// TIA Portal V16 export
// export: Created 2022-01-12T14:32:04.6959631Z, ExportSetting WithDefaults, DisplayName Totally Integrated Automation Portal, DisplayVersion V16 Update 4, DisplayName TIA Portal Version Control Interface, DisplayVersion V16 Update 2, DisplayName TIA Portal Openness, DisplayVersion V16 Update 4, DisplayName STEP 7 Professional, DisplayVersion V16 Update 4, DisplayName STEP 7 Safety, DisplayVersion V16, DisplayName WinCC Professional, DisplayVersion V16 Update 4
DATA_BLOCK "Cip"   // DB8
VERSION : 0.1
// stored: AutoNumber true, DBAccessibleFromOPCUA true, InstanceOfName FB_obsluga_obiektow, InstanceOfType FB
"FB_obsluga_obiektow"
   // VAR
   //    obiekt : Array[0..110] of "typObiekt";
   //    tor : Array[0..2] of "typFunkcjeObiektówCipu";
   //    x { ExternalAccessible := 'False'; ExternalVisible := 'False'; ExternalWritable := 'False'} : Int := 111;
   // END_VAR
BEGIN
   obiekt[0].typObiektu := 0;
   obiekt[1..11].typObiektu := 5;
   obiekt[12..13].typObiektu := 12;
   obiekt[14..20].typObiektu := 18;
   obiekt[21..22].typObiektu := 2;
   obiekt[23..30].typObiektu := 1;
   obiekt[31..32].typObiektu := 4;
   obiekt[33..41].typObiektu := 1;
   obiekt[42..44].typObiektu := 9;
   obiekt[45..49].typObiektu := 1;
   obiekt[50..53].typObiektu := 9;
   obiekt[54..58].typObiektu := 1;
   obiekt[59..62].typObiektu := 9;
   obiekt[63..68].typObiektu := 1;
   obiekt[69..71].typObiektu := 9;
   obiekt[72..78].typObiektu := 1;
   obiekt[79..82].typObiektu := 9;
   obiekt[83..87].typObiektu := 1;
   obiekt[88..90].typObiektu := 9;
   obiekt[91..93].typObiektu := 1;
   obiekt[94..96].typObiektu := 9;
   obiekt[97..98].typObiektu := 4;
   obiekt[99..100].typObiektu := 3;
   obiekt[101..105].typObiektu := 9;
   obiekt[106..107].typObiektu := 17;
   obiekt[108..110].typObiektu := 1;
   obiekt[0].nazwaObiektu := 'C2W1LL01';
   obiekt[1].nazwaObiektu := 'C2W1TT01';
   obiekt[2].nazwaObiektu := 'C2R1TT01';
   obiekt[3].nazwaObiektu := 'C2L1TT01';
   obiekt[4].nazwaObiektu := 'C2A1TT01';
   obiekt[5].nazwaObiektu := 'C2D1TT01';
   obiekt[6].nazwaObiektu := 'C2D2TT01';
   obiekt[7].nazwaObiektu := 'C2D3TT01';
   obiekt[8].nazwaObiektu := 'C211TT01';
   obiekt[9].nazwaObiektu := 'C212TT01';
   obiekt[10].nazwaObiektu := 'C201TT01';
   obiekt[11].nazwaObiektu := 'C202TT01';
   obiekt[12].nazwaObiektu := 'C212QIC01';
   obiekt[13].nazwaObiektu := 'C211QIC01';
   obiekt[14].nazwaObiektu := 'C2A1LT01';
   obiekt[15].nazwaObiektu := 'C2D1LT01';
   obiekt[16].nazwaObiektu := 'C2D2LT01';
   obiekt[17].nazwaObiektu := 'C2D3LT01';
   obiekt[18].nazwaObiektu := 'C2L1LT01';
   obiekt[19].nazwaObiektu := 'C2R1LT01';
   obiekt[20].nazwaObiektu := 'C2W1LT01';
   obiekt[21..22].nazwaObiektu := 'C202CV21';
   obiekt[23].nazwaObiektu := 'C201AV01';
   obiekt[24].nazwaObiektu := 'C201AV02';
   obiekt[25].nazwaObiektu := 'C201AV21';
   obiekt[26].nazwaObiektu := 'C202AV01';
   obiekt[27].nazwaObiektu := 'C202AV02';
   obiekt[28].nazwaObiektu := 'C202AV03';
   obiekt[29].nazwaObiektu := 'C202AV04';
   obiekt[30].nazwaObiektu := 'C202AV21';
   obiekt[31].nazwaObiektu := 'C202FC01';
   obiekt[32].nazwaObiektu := 'C201CP01';
   obiekt[33].nazwaObiektu := 'C211AV01';
   obiekt[34].nazwaObiektu := 'C212AV01';
   obiekt[35].nazwaObiektu := 'C2A1AV01';
   obiekt[36].nazwaObiektu := 'C2A1AV02';
   obiekt[37].nazwaObiektu := 'C2A1AV11';
   obiekt[38].nazwaObiektu := 'C2A1AV12';
   obiekt[39].nazwaObiektu := 'C2A1AV31';
   obiekt[40].nazwaObiektu := 'C2A1AV41';
   obiekt[41].nazwaObiektu := 'C2A1AV42';
   obiekt[42].nazwaObiektu := 'C2A1LH01';
   obiekt[43].nazwaObiektu := 'C2A1LL41';
   obiekt[44].nazwaObiektu := 'C2A1PD01';
   obiekt[45].nazwaObiektu := 'C2D1AV01';
   obiekt[46].nazwaObiektu := 'C2D1AV11';
   obiekt[47].nazwaObiektu := 'C2D1AV41';
   obiekt[48].nazwaObiektu := 'C2D1AV42';
   obiekt[49].nazwaObiektu := 'C2D1AV81';
   obiekt[50].nazwaObiektu := 'C2D1LH01';
   obiekt[51].nazwaObiektu := 'C2D1LL01';
   obiekt[52].nazwaObiektu := 'C2D1LL81';
   obiekt[53].nazwaObiektu := 'C2D1PD01';
   obiekt[54].nazwaObiektu := 'C2D2AV01';
   obiekt[55].nazwaObiektu := 'C2D2AV11';
   obiekt[56].nazwaObiektu := 'C2D2AV41';
   obiekt[57].nazwaObiektu := 'C2D2AV42';
   obiekt[58].nazwaObiektu := 'C2D2AV81';
   obiekt[59].nazwaObiektu := 'C2D2LH01';
   obiekt[60].nazwaObiektu := 'C2D2LL01';
   obiekt[61].nazwaObiektu := 'C2D2LL81';
   obiekt[62].nazwaObiektu := 'C2D2PD01';
   obiekt[63].nazwaObiektu := 'C2D3AV01';
   obiekt[64].nazwaObiektu := 'C2D3AV11';
   obiekt[65].nazwaObiektu := 'C2D3AV31';
   obiekt[66].nazwaObiektu := 'C2D3AV41';
   obiekt[67].nazwaObiektu := 'C2D3AV42';
   obiekt[68].nazwaObiektu := 'C2D3AV43';
   obiekt[69].nazwaObiektu := 'C2D3LH01';
   obiekt[70].nazwaObiektu := 'C2D3LL01';
   obiekt[71].nazwaObiektu := 'C2D3PD01';
   obiekt[72].nazwaObiektu := 'C2L1AV01';
   obiekt[73].nazwaObiektu := 'C2L1AV02';
   obiekt[74].nazwaObiektu := 'C2L1AV11';
   obiekt[75].nazwaObiektu := 'C2L1AV12';
   obiekt[76].nazwaObiektu := 'C2L1AV31';
   obiekt[77].nazwaObiektu := 'C2L1AV41';
   obiekt[78].nazwaObiektu := 'C2L1AV42';
   obiekt[79].nazwaObiektu := 'C2L1LH01';
   obiekt[80].nazwaObiektu := 'C2L1Ll01';
   obiekt[81].nazwaObiektu := 'C2L1Ll41';
   obiekt[82].nazwaObiektu := 'C2L1PD01';
   obiekt[83].nazwaObiektu := 'C2R1AV01';
   obiekt[84].nazwaObiektu := 'C2R1AV02';
   obiekt[85].nazwaObiektu := 'C2R1AV11';
   obiekt[86].nazwaObiektu := 'C2R1AV12';
   obiekt[87].nazwaObiektu := 'C2R1AV41';
   obiekt[88].nazwaObiektu := 'C2R1LH01';
   obiekt[89].nazwaObiektu := 'C2R1LL01';
   obiekt[90].nazwaObiektu := 'C2R1PD01';
   obiekt[91].nazwaObiektu := 'C2W1AV02';
   obiekt[92].nazwaObiektu := 'C2W1AV31';
   obiekt[93].nazwaObiektu := 'C2W1AV41';
   obiekt[94].nazwaObiektu := 'C2W1LH01';
   obiekt[95].nazwaObiektu := 'C2W1LL01';
   obiekt[96].nazwaObiektu := 'C2W1PD01';
   obiekt[97..98].nazwaObiektu := 'C2D1MP81';
   obiekt[99].nazwaObiektu := 'C2A1MP41';
   obiekt[100].nazwaObiektu := 'C2L1MP41';
   obiekt[101].nazwaObiektu := 'C211FV01';
   obiekt[102].nazwaObiektu := 'C212FV01';
   obiekt[103].nazwaObiektu := 'C2D1FV81';
   obiekt[104].nazwaObiektu := 'C2D2FV81';
   obiekt[105].nazwaObiektu := 'C2A1LL01';
   obiekt[106..107].nazwaObiektu := 'F100AV01';
   obiekt[108].nazwaObiektu := 'C2A1AV43';
   obiekt[109].nazwaObiektu := 'C2L1AV43';
   obiekt[110].nazwaObiektu := 'C2W1AV01';
   obiekt[0..20].procedura := 0;
   obiekt[21].procedura := 3;
   obiekt[22].procedura := 0;
   obiekt[23].procedura := 2;
   obiekt[24].procedura := 1;
   obiekt[25].procedura := 2;
   obiekt[26..28].procedura := 0;
   obiekt[29].procedura := 2;
   obiekt[30].procedura := 0;
   obiekt[31].procedura := 3;
   obiekt[32].procedura := 6;
   obiekt[33].procedura := 2;
   obiekt[34].procedura := 0;
   obiekt[35].procedura := 2;
   obiekt[36].procedura := 0;
   obiekt[37].procedura := 2;
   obiekt[38].procedura := 0;
   obiekt[39].procedura := 2;
   obiekt[40..71].procedura := 0;
   obiekt[72].procedura := 2;
   obiekt[73].procedura := 0;
   obiekt[74].procedura := 2;
   obiekt[75].procedura := 0;
   obiekt[76].procedura := 2;
   obiekt[77..91].procedura := 0;
   obiekt[92].procedura := 2;
   obiekt[93..98].procedura := 0;
   obiekt[99].procedura := 2;
   obiekt[100..109].procedura := 0;
   obiekt[110].procedura := 4;
   obiekt[0..20].inStartAuto := FALSE;
   obiekt[21].inStartAuto := TRUE;
   obiekt[22..23].inStartAuto := FALSE;
   obiekt[24..25].inStartAuto := TRUE;
   obiekt[26..30].inStartAuto := FALSE;
   obiekt[31..32].inStartAuto := TRUE;
   obiekt[33..34].inStartAuto := FALSE;
   obiekt[35].inStartAuto := TRUE;
   obiekt[36..91].inStartAuto := FALSE;
   obiekt[92].inStartAuto := TRUE;
   obiekt[93..110].inStartAuto := FALSE;
   obiekt[0..20].outStartUrządzenie := FALSE;
   obiekt[21].outStartUrządzenie := TRUE;
   obiekt[22..23].outStartUrządzenie := FALSE;
   obiekt[24..25].outStartUrządzenie := TRUE;
   obiekt[26..30].outStartUrządzenie := FALSE;
   obiekt[31..32].outStartUrządzenie := TRUE;
   obiekt[33..34].outStartUrządzenie := FALSE;
   obiekt[35].outStartUrządzenie := TRUE;
   obiekt[36..91].outStartUrządzenie := FALSE;
   obiekt[92].outStartUrządzenie := TRUE;
   obiekt[93..110].outStartUrządzenie := FALSE;
   obiekt[0..110].inLiftUp := FALSE;
   obiekt[0..110].outLiftUp := FALSE;
   obiekt[0..110].inLiftDown := FALSE;
   obiekt[0..110].outLiftDown := FALSE;
   obiekt[0..20].inZadaneWysterowanieAuto := 0.0;
   obiekt[21].inZadaneWysterowanieAuto := 100.0;
   obiekt[22..23].inZadaneWysterowanieAuto := 0.0;
   obiekt[24].inZadaneWysterowanieAuto := 100.0;
   obiekt[25..28].inZadaneWysterowanieAuto := 0.0;
   obiekt[29].inZadaneWysterowanieAuto := 100.0;
   obiekt[30].inZadaneWysterowanieAuto := 0.0;
   obiekt[31..32].inZadaneWysterowanieAuto := 100.0;
   obiekt[33..98].inZadaneWysterowanieAuto := 0.0;
   obiekt[99].inZadaneWysterowanieAuto := 100.0;
   obiekt[100..110].inZadaneWysterowanieAuto := 0.0;
   obiekt[0..20].outWysterowanieUrządzenia := 0.0;
   obiekt[21].outWysterowanieUrządzenia := 100.0;
   obiekt[22..23].outWysterowanieUrządzenia := 0.0;
   obiekt[24].outWysterowanieUrządzenia := 100.0;
   obiekt[25..30].outWysterowanieUrządzenia := 0.0;
   obiekt[31..32].outWysterowanieUrządzenia := 100.0;
   obiekt[33..110].outWysterowanieUrządzenia := 0.0;
   obiekt[0].inJestPotwWysterowania := TRUE;
   obiekt[1..22].inJestPotwWysterowania := FALSE;
   obiekt[23..24].inJestPotwWysterowania := TRUE;
   obiekt[25].inJestPotwWysterowania := FALSE;
   obiekt[26..29].inJestPotwWysterowania := TRUE;
   obiekt[30].inJestPotwWysterowania := FALSE;
   obiekt[31..40].inJestPotwWysterowania := TRUE;
   obiekt[41].inJestPotwWysterowania := FALSE;
   obiekt[42..48].inJestPotwWysterowania := TRUE;
   obiekt[49].inJestPotwWysterowania := FALSE;
   obiekt[50..57].inJestPotwWysterowania := TRUE;
   obiekt[58].inJestPotwWysterowania := FALSE;
   obiekt[59..77].inJestPotwWysterowania := TRUE;
   obiekt[78].inJestPotwWysterowania := FALSE;
   obiekt[79..98].inJestPotwWysterowania := TRUE;
   obiekt[99..100].inJestPotwWysterowania := FALSE;
   obiekt[101..105].inJestPotwWysterowania := TRUE;
   obiekt[106..109].inJestPotwWysterowania := FALSE;
   obiekt[110].inJestPotwWysterowania := TRUE;
   obiekt[0..20].diPotwWysterowania := FALSE;
   obiekt[21].diPotwWysterowania := TRUE;
   obiekt[22..41].diPotwWysterowania := FALSE;
   obiekt[42].diPotwWysterowania := TRUE;
   obiekt[43..49].diPotwWysterowania := FALSE;
   obiekt[50].diPotwWysterowania := TRUE;
   obiekt[51..58].diPotwWysterowania := FALSE;
   obiekt[59].diPotwWysterowania := TRUE;
   obiekt[60..68].diPotwWysterowania := FALSE;
   obiekt[69].diPotwWysterowania := TRUE;
   obiekt[70..77].diPotwWysterowania := FALSE;
   obiekt[78..79].diPotwWysterowania := TRUE;
   obiekt[80..87].diPotwWysterowania := FALSE;
   obiekt[88].diPotwWysterowania := TRUE;
   obiekt[89..93].diPotwWysterowania := FALSE;
   obiekt[94].diPotwWysterowania := TRUE;
   obiekt[95..110].diPotwWysterowania := FALSE;
   obiekt[0..110].inJestPotwNiewysterowania := FALSE;
   obiekt[0..21].diPotwNieWysterowania := FALSE;
   obiekt[22].diPotwNieWysterowania := TRUE;
   obiekt[23..110].diPotwNieWysterowania := FALSE;
   obiekt[0..20].inZezwolenieNaPracę := FALSE;
   obiekt[21..41].inZezwolenieNaPracę := TRUE;
   obiekt[42..44].inZezwolenieNaPracę := FALSE;
   obiekt[45..49].inZezwolenieNaPracę := TRUE;
   obiekt[50..53].inZezwolenieNaPracę := FALSE;
   obiekt[54..58].inZezwolenieNaPracę := TRUE;
   obiekt[59..62].inZezwolenieNaPracę := FALSE;
   obiekt[63..68].inZezwolenieNaPracę := TRUE;
   obiekt[69..71].inZezwolenieNaPracę := FALSE;
   obiekt[72..78].inZezwolenieNaPracę := TRUE;
   obiekt[79..82].inZezwolenieNaPracę := FALSE;
   obiekt[83..87].inZezwolenieNaPracę := TRUE;
   obiekt[88..90].inZezwolenieNaPracę := FALSE;
   obiekt[91..93].inZezwolenieNaPracę := TRUE;
   obiekt[94..96].inZezwolenieNaPracę := FALSE;
   obiekt[97..100].inZezwolenieNaPracę := TRUE;
   obiekt[101..107].inZezwolenieNaPracę := FALSE;
   obiekt[108..110].inZezwolenieNaPracę := TRUE;
   obiekt[0..110].Awaria := FALSE;
   obiekt[0..110].ResetAwaria := FALSE;
   obiekt[0..110].kodBłedu := 16#0000;
   obiekt[0..110].czasDoAwariiSP := 1000;
   obiekt[0..30].czasDoAwariiPV := 0;
   obiekt[31].czasDoAwariiPV := 17;
   obiekt[32..41].czasDoAwariiPV := 0;
   obiekt[42].czasDoAwariiPV := 5;
   obiekt[43..49].czasDoAwariiPV := 0;
   obiekt[50].czasDoAwariiPV := 5;
   obiekt[51..58].czasDoAwariiPV := 0;
   obiekt[59].czasDoAwariiPV := 5;
   obiekt[60..68].czasDoAwariiPV := 0;
   obiekt[69].czasDoAwariiPV := 5;
   obiekt[70..78].czasDoAwariiPV := 0;
   obiekt[79].czasDoAwariiPV := 5;
   obiekt[80..87].czasDoAwariiPV := 0;
   obiekt[88].czasDoAwariiPV := 5;
   obiekt[89..93].czasDoAwariiPV := 0;
   obiekt[94].czasDoAwariiPV := 5;
   obiekt[95..110].czasDoAwariiPV := 0;
   obiekt[0..110].czasPracyGodziny := 0.0;
   obiekt[0..110]._ := FALSE;
   obiekt[0..110].hmiPokażStacyjkę := FALSE;
   obiekt[0].hmiStanUrządzenia := 2;
   obiekt[1..20].hmiStanUrządzenia := 1;
   obiekt[21].hmiStanUrządzenia := 3;
   obiekt[22..23].hmiStanUrządzenia := 1;
   obiekt[24..25].hmiStanUrządzenia := 3;
   obiekt[26..30].hmiStanUrządzenia := 1;
   obiekt[31..32].hmiStanUrządzenia := 3;
   obiekt[33..34].hmiStanUrządzenia := 1;
   obiekt[35].hmiStanUrządzenia := 3;
   obiekt[36..41].hmiStanUrządzenia := 1;
   obiekt[42].hmiStanUrządzenia := 3;
   obiekt[43..49].hmiStanUrządzenia := 1;
   obiekt[50].hmiStanUrządzenia := 3;
   obiekt[51..58].hmiStanUrządzenia := 1;
   obiekt[59].hmiStanUrządzenia := 3;
   obiekt[60..68].hmiStanUrządzenia := 1;
   obiekt[69].hmiStanUrządzenia := 3;
   obiekt[70..78].hmiStanUrządzenia := 1;
   obiekt[79].hmiStanUrządzenia := 3;
   obiekt[80].hmiStanUrządzenia := 4;
   obiekt[81..87].hmiStanUrządzenia := 1;
   obiekt[88].hmiStanUrządzenia := 2;
   obiekt[89].hmiStanUrządzenia := 4;
   obiekt[90..91].hmiStanUrządzenia := 1;
   obiekt[92].hmiStanUrządzenia := 3;
   obiekt[93].hmiStanUrządzenia := 1;
   obiekt[94..95].hmiStanUrządzenia := 2;
   obiekt[96..104].hmiStanUrządzenia := 1;
   obiekt[105].hmiStanUrządzenia := 4;
   obiekt[106..110].hmiStanUrządzenia := 1;
   obiekt[0..110].hmiTrybAutoManual := FALSE;
   obiekt[0..110].hmiManualStart := FALSE;
   obiekt[0..110].hmiManualStop := FALSE;
   obiekt[0..110].hmiManualLiftUp := FALSE;
   obiekt[0..110].hmiManualLiftDown := FALSE;
   obiekt[0..110].hmiManualneWysterowanie := 0.0;
   obiekt[0].hmiSymulujSygnałyWejsciowe := TRUE;
   obiekt[1..7].hmiSymulujSygnałyWejsciowe := FALSE;
   obiekt[8].hmiSymulujSygnałyWejsciowe := TRUE;
   obiekt[9].hmiSymulujSygnałyWejsciowe := FALSE;
   obiekt[10].hmiSymulujSygnałyWejsciowe := TRUE;
   obiekt[11..12].hmiSymulujSygnałyWejsciowe := FALSE;
   obiekt[13].hmiSymulujSygnałyWejsciowe := TRUE;
   obiekt[14..23].hmiSymulujSygnałyWejsciowe := FALSE;
   obiekt[24].hmiSymulujSygnałyWejsciowe := TRUE;
   obiekt[25..31].hmiSymulujSygnałyWejsciowe := FALSE;
   obiekt[32..33].hmiSymulujSygnałyWejsciowe := TRUE;
   obiekt[34].hmiSymulujSygnałyWejsciowe := FALSE;
   obiekt[35].hmiSymulujSygnałyWejsciowe := TRUE;
   obiekt[36].hmiSymulujSygnałyWejsciowe := FALSE;
   obiekt[37].hmiSymulujSygnałyWejsciowe := TRUE;
   obiekt[38..39].hmiSymulujSygnałyWejsciowe := FALSE;
   obiekt[40].hmiSymulujSygnałyWejsciowe := TRUE;
   obiekt[41..71].hmiSymulujSygnałyWejsciowe := FALSE;
   obiekt[72].hmiSymulujSygnałyWejsciowe := TRUE;
   obiekt[73].hmiSymulujSygnałyWejsciowe := FALSE;
   obiekt[74].hmiSymulujSygnałyWejsciowe := TRUE;
   obiekt[75].hmiSymulujSygnałyWejsciowe := FALSE;
   obiekt[76..77].hmiSymulujSygnałyWejsciowe := TRUE;
   obiekt[78..79].hmiSymulujSygnałyWejsciowe := FALSE;
   obiekt[80].hmiSymulujSygnałyWejsciowe := TRUE;
   obiekt[81..82].hmiSymulujSygnałyWejsciowe := FALSE;
   obiekt[83].hmiSymulujSygnałyWejsciowe := TRUE;
   obiekt[84].hmiSymulujSygnałyWejsciowe := FALSE;
   obiekt[85].hmiSymulujSygnałyWejsciowe := TRUE;
   obiekt[86].hmiSymulujSygnałyWejsciowe := FALSE;
   obiekt[87..89].hmiSymulujSygnałyWejsciowe := TRUE;
   obiekt[90..91].hmiSymulujSygnałyWejsciowe := FALSE;
   obiekt[92..95].hmiSymulujSygnałyWejsciowe := TRUE;
   obiekt[96..104].hmiSymulujSygnałyWejsciowe := FALSE;
   obiekt[105..106].hmiSymulujSygnałyWejsciowe := TRUE;
   obiekt[107..109].hmiSymulujSygnałyWejsciowe := FALSE;
   obiekt[110].hmiSymulujSygnałyWejsciowe := TRUE;
   obiekt[0..79].hmiSymulacjaPotwWysterowania := FALSE;
   obiekt[80].hmiSymulacjaPotwWysterowania := TRUE;
   obiekt[81..88].hmiSymulacjaPotwWysterowania := FALSE;
   obiekt[89].hmiSymulacjaPotwWysterowania := TRUE;
   obiekt[90..104].hmiSymulacjaPotwWysterowania := FALSE;
   obiekt[105].hmiSymulacjaPotwWysterowania := TRUE;
   obiekt[106..110].hmiSymulacjaPotwWysterowania := FALSE;
   obiekt[0..110].hmiSymulacjaPotwNieWysterowania := FALSE;
   obiekt[0..7].hmiSymulowanaWartośćAnalogowa := 0.0;
   obiekt[8].hmiSymulowanaWartośćAnalogowa := 45.0;
   obiekt[9].hmiSymulowanaWartośćAnalogowa := 0.0;
   obiekt[10].hmiSymulowanaWartośćAnalogowa := 19.0;
   obiekt[11..105].hmiSymulowanaWartośćAnalogowa := 0.0;
   obiekt[106].hmiSymulowanaWartośćAnalogowa := 5.0;
   obiekt[107..110].hmiSymulowanaWartośćAnalogowa := 0.0;
   obiekt[0..23].hmiPotwNieWysterowania := TRUE;
   obiekt[24..25].hmiPotwNieWysterowania := FALSE;
   obiekt[26..30].hmiPotwNieWysterowania := TRUE;
   obiekt[31..32].hmiPotwNieWysterowania := FALSE;
   obiekt[33..34].hmiPotwNieWysterowania := TRUE;
   obiekt[35].hmiPotwNieWysterowania := FALSE;
   obiekt[36..91].hmiPotwNieWysterowania := TRUE;
   obiekt[92].hmiPotwNieWysterowania := FALSE;
   obiekt[93..110].hmiPotwNieWysterowania := TRUE;
   obiekt[0..23].hmiPotwWysterowania := FALSE;
   obiekt[24..25].hmiPotwWysterowania := TRUE;
   obiekt[26..31].hmiPotwWysterowania := FALSE;
   obiekt[32].hmiPotwWysterowania := TRUE;
   obiekt[33..34].hmiPotwWysterowania := FALSE;
   obiekt[35].hmiPotwWysterowania := TRUE;
   obiekt[36..41].hmiPotwWysterowania := FALSE;
   obiekt[42].hmiPotwWysterowania := TRUE;
   obiekt[43..49].hmiPotwWysterowania := FALSE;
   obiekt[50].hmiPotwWysterowania := TRUE;
   obiekt[51..58].hmiPotwWysterowania := FALSE;
   obiekt[59].hmiPotwWysterowania := TRUE;
   obiekt[60..68].hmiPotwWysterowania := FALSE;
   obiekt[69].hmiPotwWysterowania := TRUE;
   obiekt[70..78].hmiPotwWysterowania := FALSE;
   obiekt[79..80].hmiPotwWysterowania := TRUE;
   obiekt[81..88].hmiPotwWysterowania := FALSE;
   obiekt[89].hmiPotwWysterowania := TRUE;
   obiekt[90..91].hmiPotwWysterowania := FALSE;
   obiekt[92].hmiPotwWysterowania := TRUE;
   obiekt[93..104].hmiPotwWysterowania := FALSE;
   obiekt[105].hmiPotwWysterowania := TRUE;
   obiekt[106..110].hmiPotwWysterowania := FALSE;
   obiekt[0..30].hmiZasilanieOK := FALSE;
   obiekt[31..32].hmiZasilanieOK := TRUE;
   obiekt[33..98].hmiZasilanieOK := FALSE;
   obiekt[99..100].hmiZasilanieOK := TRUE;
   obiekt[101..110].hmiZasilanieOK := FALSE;
   obiekt[0..110].hmiResetAwaria := FALSE;
   obiekt[0..110].hmiPrądFalownika := 0.0;
   obiekt[0..110].___ := FALSE;
   obiekt[0..110].inPomiarRaw := 0;
   obiekt[0..110].minSkali := -50.0;
   obiekt[0..12].maxskali := 150.0;
   obiekt[13].maxskali := 50.0;
   obiekt[14..110].maxskali := 150.0;
   obiekt[0..110].tFiltr := 0.9;
   obiekt[0].pomiarTymczas := 0.0;
   obiekt[1..20].pomiarTymczas := -50.0;
   obiekt[21..110].pomiarTymczas := 0.0;
   obiekt[0].wyjTymczas := 0.0;
   obiekt[1..7].wyjTymczas := -49.99997;
   obiekt[8].wyjTymczas := 35.5;
   obiekt[9].wyjTymczas := -49.99997;
   obiekt[10].wyjTymczas := 12.1;
   obiekt[11..20].wyjTymczas := -49.99997;
   obiekt[21..105].wyjTymczas := 0.0;
   obiekt[106].wyjTymczas := 4.5;
   obiekt[107..110].wyjTymczas := 0.0;
   obiekt[0].WartośćPomiaru := 0.0;
   obiekt[1..7].WartośćPomiaru := -49.99997;
   obiekt[8].WartośćPomiaru := 45.0;
   obiekt[9].WartośćPomiaru := -49.99997;
   obiekt[10].WartośćPomiaru := 19.0;
   obiekt[11..12].WartośćPomiaru := -49.99997;
   obiekt[13].WartośćPomiaru := 0.0;
   obiekt[14..20].WartośćPomiaru := -49.99997;
   obiekt[21..105].WartośćPomiaru := 0.0;
   obiekt[106].WartośćPomiaru := 5.0;
   obiekt[107..110].WartośćPomiaru := 0.0;
   obiekt[0..110].____ := FALSE;
   obiekt[0].hmiMetry3NaImpuls := 0.01;
   obiekt[1..105].hmiMetry3NaImpuls := 0.001;
   obiekt[106].hmiMetry3NaImpuls := 6.944445E-05;
   obiekt[107].hmiMetry3NaImpuls := 0.0;
   obiekt[108..110].hmiMetry3NaImpuls := 0.001;
   obiekt[0..110].diImpulsy := FALSE;
   obiekt[0..110].R_Trig := FALSE;
   obiekt[0..105].startLicznik1 := FALSE;
   obiekt[106].startLicznik1 := TRUE;
   obiekt[107..110].startLicznik1 := FALSE;
   obiekt[0..110].zerujLicznik1 := FALSE;
   obiekt[0..110].startLicznik2 := FALSE;
   obiekt[0..110].zerujLicznik2 := FALSE;
   obiekt[0..110].startLicznik3 := FALSE;
   obiekt[0..110].zerujLicznik3 := FALSE;
   obiekt[0..105].licznik1 := 0.0;
   obiekt[106].licznik1 := 0.05576352;
   obiekt[107..110].licznik1 := 0.0;
   obiekt[0..110].licznik2 := 0.0;
   obiekt[0..110].licznik3 := 0.0;
   obiekt[0..110].licznikTotalImpulsy := 0;
   obiekt[0..110].Lreal_1 := 0.0;
   obiekt[0..110].Lreal_2 := 0.0;
   obiekt[0..110]._____ := FALSE;
   obiekt[0..20].pid_SP := 0.0;
   obiekt[21].pid_SP := 60.0;
   obiekt[22..31].pid_SP := 0.0;
   obiekt[32].pid_SP := 15.0;
   obiekt[33..110].pid_SP := 0.0;
   obiekt[0..20].pid_PV := 0.0;
   obiekt[21].pid_PV := 19.0;
   obiekt[22..31].pid_PV := 0.0;
   obiekt[32].pid_PV := 5.0;
   obiekt[33..110].pid_PV := 0.0;
   obiekt[0..110].pid_P := 1.0;
   obiekt[0..110].pid_I := 10.0;
   obiekt[0..110].pid_D := 0.0;
   obiekt[0..11].pid_Rampa := 1.0;
   obiekt[12..13].pid_Rampa := -49.99997;
   obiekt[14..110].pid_Rampa := 1.0;
   obiekt[0..20].pid_Out := 0.0;
   obiekt[21].pid_Out := 100.0;
   obiekt[22..31].pid_Out := 0.0;
   obiekt[32].pid_Out := 100.0;
   obiekt[33..110].pid_Out := 0.0;
   obiekt[0..110].______ := FALSE;
   obiekt[0..20].SetReset.inSet := FALSE;
   obiekt[21].SetReset.inSet := TRUE;
   obiekt[22..24].SetReset.inSet := FALSE;
   obiekt[25].SetReset.inSet := TRUE;
   obiekt[26..30].SetReset.inSet := FALSE;
   obiekt[31].SetReset.inSet := TRUE;
   obiekt[32..34].SetReset.inSet := FALSE;
   obiekt[35].SetReset.inSet := TRUE;
   obiekt[36..84].SetReset.inSet := FALSE;
   obiekt[85].SetReset.inSet := TRUE;
   obiekt[86..91].SetReset.inSet := FALSE;
   obiekt[92].SetReset.inSet := TRUE;
   obiekt[93..110].SetReset.inSet := FALSE;
   obiekt[0].SetReset.inReset := TRUE;
   obiekt[1..22].SetReset.inReset := FALSE;
   obiekt[23].SetReset.inReset := TRUE;
   obiekt[24..28].SetReset.inReset := FALSE;
   obiekt[29].SetReset.inReset := TRUE;
   obiekt[30..31].SetReset.inReset := FALSE;
   obiekt[32..33].SetReset.inReset := TRUE;
   obiekt[34..36].SetReset.inReset := FALSE;
   obiekt[37].SetReset.inReset := TRUE;
   obiekt[38].SetReset.inReset := FALSE;
   obiekt[39].SetReset.inReset := TRUE;
   obiekt[40..71].SetReset.inReset := FALSE;
   obiekt[72].SetReset.inReset := TRUE;
   obiekt[73].SetReset.inReset := FALSE;
   obiekt[74].SetReset.inReset := TRUE;
   obiekt[75].SetReset.inReset := FALSE;
   obiekt[76].SetReset.inReset := TRUE;
   obiekt[77..82].SetReset.inReset := FALSE;
   obiekt[83].SetReset.inReset := TRUE;
   obiekt[84..98].SetReset.inReset := FALSE;
   obiekt[99].SetReset.inReset := TRUE;
   obiekt[100..109].SetReset.inReset := FALSE;
   obiekt[110].SetReset.inReset := TRUE;
   obiekt[0].SetReset.czasDoSet := 1;
   obiekt[1..20].SetReset.czasDoSet := 0;
   obiekt[21].SetReset.czasDoSet := 2;
   obiekt[22].SetReset.czasDoSet := 0;
   obiekt[23].SetReset.czasDoSet := 2;
   obiekt[24].SetReset.czasDoSet := 0;
   obiekt[25].SetReset.czasDoSet := 2;
   obiekt[26..28].SetReset.czasDoSet := 0;
   obiekt[29].SetReset.czasDoSet := 10;
   obiekt[30].SetReset.czasDoSet := 0;
   obiekt[31..32].SetReset.czasDoSet := 3;
   obiekt[33].SetReset.czasDoSet := 2;
   obiekt[34].SetReset.czasDoSet := 0;
   obiekt[35].SetReset.czasDoSet := 3;
   obiekt[36].SetReset.czasDoSet := 0;
   obiekt[37].SetReset.czasDoSet := 1;
   obiekt[38].SetReset.czasDoSet := 0;
   obiekt[39].SetReset.czasDoSet := 1;
   obiekt[40..71].SetReset.czasDoSet := 0;
   obiekt[72].SetReset.czasDoSet := 3;
   obiekt[73].SetReset.czasDoSet := 0;
   obiekt[74].SetReset.czasDoSet := 1;
   obiekt[75].SetReset.czasDoSet := 0;
   obiekt[76].SetReset.czasDoSet := 1;
   obiekt[77..82].SetReset.czasDoSet := 0;
   obiekt[83].SetReset.czasDoSet := 3;
   obiekt[84].SetReset.czasDoSet := 0;
   obiekt[85].SetReset.czasDoSet := 1;
   obiekt[86..91].SetReset.czasDoSet := 0;
   obiekt[92].SetReset.czasDoSet := 1;
   obiekt[93..98].SetReset.czasDoSet := 0;
   obiekt[99].SetReset.czasDoSet := 10;
   obiekt[100..109].SetReset.czasDoSet := 0;
   obiekt[110].SetReset.czasDoSet := 1;
   obiekt[0].SetReset.czasDoReset := 5;
   obiekt[1..20].SetReset.czasDoReset := 0;
   obiekt[21].SetReset.czasDoReset := 2;
   obiekt[22].SetReset.czasDoReset := 0;
   obiekt[23].SetReset.czasDoReset := 2;
   obiekt[24].SetReset.czasDoReset := 0;
   obiekt[25].SetReset.czasDoReset := 2;
   obiekt[26..30].SetReset.czasDoReset := 0;
   obiekt[31].SetReset.czasDoReset := 60;
   obiekt[32].SetReset.czasDoReset := 5;
   obiekt[33].SetReset.czasDoReset := 2;
   obiekt[34].SetReset.czasDoReset := 0;
   obiekt[35].SetReset.czasDoReset := 10;
   obiekt[36].SetReset.czasDoReset := 0;
   obiekt[37].SetReset.czasDoReset := 1;
   obiekt[38].SetReset.czasDoReset := 0;
   obiekt[39].SetReset.czasDoReset := 5;
   obiekt[40..71].SetReset.czasDoReset := 0;
   obiekt[72].SetReset.czasDoReset := 10;
   obiekt[73].SetReset.czasDoReset := 0;
   obiekt[74].SetReset.czasDoReset := 1;
   obiekt[75].SetReset.czasDoReset := 0;
   obiekt[76].SetReset.czasDoReset := 5;
   obiekt[77..82].SetReset.czasDoReset := 0;
   obiekt[83].SetReset.czasDoReset := 10;
   obiekt[84].SetReset.czasDoReset := 0;
   obiekt[85].SetReset.czasDoReset := 1;
   obiekt[86..109].SetReset.czasDoReset := 0;
   obiekt[110].SetReset.czasDoReset := 5;
   obiekt[0..20].SetReset.wyjście := FALSE;
   obiekt[21].SetReset.wyjście := TRUE;
   obiekt[22..24].SetReset.wyjście := FALSE;
   obiekt[25].SetReset.wyjście := TRUE;
   obiekt[26..30].SetReset.wyjście := FALSE;
   obiekt[31].SetReset.wyjście := TRUE;
   obiekt[32..34].SetReset.wyjście := FALSE;
   obiekt[35].SetReset.wyjście := TRUE;
   obiekt[36..91].SetReset.wyjście := FALSE;
   obiekt[92].SetReset.wyjście := TRUE;
   obiekt[93..110].SetReset.wyjście := FALSE;
   obiekt[0..20].SetReset.setCzas := 0;
   obiekt[21].SetReset.setCzas := 2;
   obiekt[22..24].SetReset.setCzas := 0;
   obiekt[25].SetReset.setCzas := 2;
   obiekt[26..30].SetReset.setCzas := 0;
   obiekt[31].SetReset.setCzas := 3;
   obiekt[32..34].SetReset.setCzas := 0;
   obiekt[35].SetReset.setCzas := 3;
   obiekt[36..91].SetReset.setCzas := 0;
   obiekt[92].SetReset.setCzas := 1;
   obiekt[93..110].SetReset.setCzas := 0;
   obiekt[0..20].SetReset.resetCzas := 1;
   obiekt[21].SetReset.resetCzas := 3;
   obiekt[22].SetReset.resetCzas := 1;
   obiekt[23].SetReset.resetCzas := 0;
   obiekt[24].SetReset.resetCzas := 1;
   obiekt[25].SetReset.resetCzas := 3;
   obiekt[26..28].SetReset.resetCzas := 1;
   obiekt[29].SetReset.resetCzas := 0;
   obiekt[30].SetReset.resetCzas := 1;
   obiekt[31].SetReset.resetCzas := 61;
   obiekt[32..33].SetReset.resetCzas := 0;
   obiekt[34].SetReset.resetCzas := 1;
   obiekt[35].SetReset.resetCzas := 11;
   obiekt[36].SetReset.resetCzas := 1;
   obiekt[37].SetReset.resetCzas := 0;
   obiekt[38].SetReset.resetCzas := 1;
   obiekt[39].SetReset.resetCzas := 0;
   obiekt[40..71].SetReset.resetCzas := 1;
   obiekt[72].SetReset.resetCzas := 0;
   obiekt[73].SetReset.resetCzas := 1;
   obiekt[74].SetReset.resetCzas := 0;
   obiekt[75].SetReset.resetCzas := 1;
   obiekt[76].SetReset.resetCzas := 0;
   obiekt[77..98].SetReset.resetCzas := 1;
   obiekt[99].SetReset.resetCzas := 0;
   obiekt[100..109].SetReset.resetCzas := 1;
   obiekt[110].SetReset.resetCzas := 0;
   obiekt[0..110].Flipaj.in := FALSE;
   obiekt[0..110].Flipaj.start_od_zera := FALSE;
   obiekt[0..110].Flipaj.Q := FALSE;
   obiekt[0..110].Flipaj.ile_petli := 0;
   obiekt[0..110].Flipaj.czas_ON := 0;
   obiekt[0..110].Flipaj.czas_OFF := 0;
   obiekt[0..110].Flipaj.licznik_petli := 1;
   obiekt[0..110].Flipaj.licznik := 0;
   obiekt[0..110].I1 := 0;
   obiekt[0..110].l2 := 0.0;
   obiekt[0..110].l4 := 16#0000;
   tor[0..2]."-na stacji CIP duże zbiorniki i zawory pod nimi" := FALSE;
   tor[0].pompaPodawaniaCip := 0;
   tor[1].pompaPodawaniaCip := 32;
   tor[2].pompaPodawaniaCip := 31;
   tor[0].zawórZrzutowyDoKanalizacji := 0;
   tor[1].zawórZrzutowyDoKanalizacji := 33;
   tor[2].zawórZrzutowyDoKanalizacji := 34;
   tor[0].zawórWydawczyCip := 0;
   tor[1].zawórWydawczyCip := 24;
   tor[2].zawórWydawczyCip := 27;
   tor[0].zawórBypassPrzygotowaniaStacji := 0;
   tor[1].zawórBypassPrzygotowaniaStacji := 23;
   tor[2].zawórBypassPrzygotowaniaStacji := 26;
   tor[0].zawórParowyOdcinający := 0;
   tor[1].zawórParowyOdcinający := 25;
   tor[2].zawórParowyOdcinający := 30;
   tor[0].zawórParowyRegulacyjny := 0;
   tor[1].zawórParowyRegulacyjny := 21;
   tor[2].zawórParowyRegulacyjny := 22;
   tor[0].zawórWydawczyWodyWtórnej := 0;
   tor[1].zawórWydawczyWodyWtórnej := 83;
   tor[2].zawórWydawczyWodyWtórnej := 84;
   tor[0].zawórPowrotnyWodyWtórnej := 0;
   tor[1].zawórPowrotnyWodyWtórnej := 85;
   tor[2].zawórPowrotnyWodyWtórnej := 86;
   tor[0].zawórWydawczyŁugu := 0;
   tor[1].zawórWydawczyŁugu := 72;
   tor[2].zawórWydawczyŁugu := 73;
   tor[0].zawórPowrotnyŁugu := 0;
   tor[1].zawórPowrotnyŁugu := 74;
   tor[2].zawórPowrotnyŁugu := 75;
   tor[0].zawórWydawczyKwasu := 0;
   tor[1].zawórWydawczyKwasu := 35;
   tor[2].zawórWydawczyKwasu := 36;
   tor[0].zawórPowrotnyKwasu := 0;
   tor[1].zawórPowrotnyKwasu := 37;
   tor[2].zawórPowrotnyKwasu := 38;
   tor[0].zawórWydawczyWodyCzystej := 0;
   tor[1].zawórWydawczyWodyCzystej := 110;
   tor[2].zawórWydawczyWodyCzystej := 91;
   tor[0].zawórWydawczyDezynfekantu := 0;
   tor[1].zawórWydawczyDezynfekantu := 45;
   tor[2].zawórWydawczyDezynfekantu := 54;
   tor[0].zawórWydawczyDezynfekantu_2 := 0;
   tor[1].zawórWydawczyDezynfekantu_2 := 63;
   tor[2].zawórWydawczyDezynfekantu_2 := 0;
   tor[0].zawórPowrotnyDezynfekantu := 0;
   tor[1].zawórPowrotnyDezynfekantu := 46;
   tor[2].zawórPowrotnyDezynfekantu := 55;
   tor[0].zawórPowrotnyDezynfekantu_2 := 0;
   tor[1].zawórPowrotnyDezynfekantu_2 := 64;
   tor[2].zawórPowrotnyDezynfekantu_2 := 0;
   tor[0].zawórStopowyPowrotuDezynfekantu := 0;
   tor[1].zawórStopowyPowrotuDezynfekantu := 47;
   tor[2].zawórStopowyPowrotuDezynfekantu := 56;
   tor[0].zawórStopowyPowrotuDezynfekantu_2 := 0;
   tor[1].zawórStopowyPowrotuDezynfekantu_2 := 66;
   tor[2].zawórStopowyPowrotuDezynfekantu_2 := 0;
   tor[0].zawórNaGruszkęZbiornikaŁugu := 0;
   tor[1].zawórNaGruszkęZbiornikaŁugu := 77;
   tor[2].zawórNaGruszkęZbiornikaŁugu := 0;
   tor[0].zawórNaGruszkęZbiornikaKwasu := 0;
   tor[1].zawórNaGruszkęZbiornikaKwasu := 40;
   tor[2].zawórNaGruszkęZbiornikaKwasu := 0;
   tor[0].zawórNaGruszkęZbiornikaWodyWtórnej := 0;
   tor[1].zawórNaGruszkęZbiornikaWodyWtórnej := 87;
   tor[2].zawórNaGruszkęZbiornikaWodyWtórnej := 0;
   tor[0].zawórNaGruszkęZbiornikaWodyCzystej := 0;
   tor[1].zawórNaGruszkęZbiornikaWodyCzystej := 93;
   tor[2].zawórNaGruszkęZbiornikaWodyCzystej := 0;
   tor[0].zawórNaGruszkęZbiornikaDezynfekantu := 0;
   tor[1].zawórNaGruszkęZbiornikaDezynfekantu := 48;
   tor[2].zawórNaGruszkęZbiornikaDezynfekantu := 57;
   tor[0].zawórNaGruszkęZbiornikaDezynfekantu_2 := 0;
   tor[1].zawórNaGruszkęZbiornikaDezynfekantu_2 := 67;
   tor[2].zawórNaGruszkęZbiornikaDezynfekantu_2 := 0;
   tor[0].zawórWodaNaGruszkęZbiornikaDezynfekantu_2 := 0;
   tor[1].zawórWodaNaGruszkęZbiornikaDezynfekantu_2 := 68;
   tor[2].zawórWodaNaGruszkęZbiornikaDezynfekantu_2 := 0;
   tor[0..1].zawórUzupełnianiaWodyCzystejZbŁugu := 76;
   tor[2].zawórUzupełnianiaWodyCzystejZbŁugu := 0;
   tor[0..1].zawórUzupełnianiaWodyCzystejZbKwasu := 39;
   tor[2].zawórUzupełnianiaWodyCzystejZbKwasu := 0;
   tor[0..2].zawórUzupełnianiaWodyCzystejZbWodyWtórnej := 0;
   tor[0..1].zawórUzupełnianiaWodyCzystejZbWodyCzystej := 92;
   tor[2].zawórUzupełnianiaWodyCzystejZbWodyCzystej := 0;
   tor[0..2].ZawórUzupełnianiaWodyCzystejZbDezynfekantu := 0;
   tor[0].ZawórUzupełnianiaWodyCzystejZbDezynfekantu_2 := 0;
   tor[1].ZawórUzupełnianiaWodyCzystejZbDezynfekantu_2 := 65;
   tor[2].ZawórUzupełnianiaWodyCzystejZbDezynfekantu_2 := 0;
   tor[0..2]."---zbiorniki główne na stacji CIP -czujniki" := FALSE;
   tor[0].zbiornikŁugu.czujnikDolnegoPoziomu := 80;
   tor[1..2].zbiornikŁugu.czujnikDolnegoPoziomu := 0;
   tor[0].zbiornikŁugu.czujnikGórnegoPoziomu := 79;
   tor[1..2].zbiornikŁugu.czujnikGórnegoPoziomu := 0;
   tor[0].zbiornikŁugu.temperatura := 3;
   tor[1..2].zbiornikŁugu.temperatura := 0;
   tor[0].zbiornikŁugu.poziomAnalogowy := 18;
   tor[1..2].zbiornikŁugu.poziomAnalogowy := 0;
   tor[0].zbiornikŁugu.czujnikwłazu := 82;
   tor[1..2].zbiornikŁugu.czujnikwłazu := 0;
   tor[0].zbiornikKwasu.czujnikDolnegoPoziomu := 105;
   tor[1..2].zbiornikKwasu.czujnikDolnegoPoziomu := 0;
   tor[0].zbiornikKwasu.czujnikGórnegoPoziomu := 42;
   tor[1..2].zbiornikKwasu.czujnikGórnegoPoziomu := 0;
   tor[0].zbiornikKwasu.temperatura := 4;
   tor[1..2].zbiornikKwasu.temperatura := 0;
   tor[0].zbiornikKwasu.poziomAnalogowy := 14;
   tor[1..2].zbiornikKwasu.poziomAnalogowy := 0;
   tor[0].zbiornikKwasu.czujnikwłazu := 44;
   tor[1..2].zbiornikKwasu.czujnikwłazu := 0;
   tor[0].zbiornikWodyWtórnej.czujnikDolnegoPoziomu := 89;
   tor[1..2].zbiornikWodyWtórnej.czujnikDolnegoPoziomu := 0;
   tor[0].zbiornikWodyWtórnej.czujnikGórnegoPoziomu := 88;
   tor[1..2].zbiornikWodyWtórnej.czujnikGórnegoPoziomu := 0;
   tor[0].zbiornikWodyWtórnej.temperatura := 2;
   tor[1..2].zbiornikWodyWtórnej.temperatura := 0;
   tor[0].zbiornikWodyWtórnej.poziomAnalogowy := 19;
   tor[1..2].zbiornikWodyWtórnej.poziomAnalogowy := 0;
   tor[0].zbiornikWodyWtórnej.czujnikwłazu := 90;
   tor[1..2].zbiornikWodyWtórnej.czujnikwłazu := 0;
   tor[0].zbiornikwodyCzystej.czujnikDolnegoPoziomu := 95;
   tor[1..2].zbiornikwodyCzystej.czujnikDolnegoPoziomu := 0;
   tor[0].zbiornikwodyCzystej.czujnikGórnegoPoziomu := 94;
   tor[1..2].zbiornikwodyCzystej.czujnikGórnegoPoziomu := 0;
   tor[0].zbiornikwodyCzystej.temperatura := 1;
   tor[1..2].zbiornikwodyCzystej.temperatura := 0;
   tor[0].zbiornikwodyCzystej.poziomAnalogowy := 20;
   tor[1..2].zbiornikwodyCzystej.poziomAnalogowy := 0;
   tor[0].zbiornikwodyCzystej.czujnikwłazu := 96;
   tor[1..2].zbiornikwodyCzystej.czujnikwłazu := 0;
   tor[0].zbiornikDezynfekantu.czujnikDolnegoPoziomu := 0;
   tor[1].zbiornikDezynfekantu.czujnikDolnegoPoziomu := 51;
   tor[2].zbiornikDezynfekantu.czujnikDolnegoPoziomu := 60;
   tor[0].zbiornikDezynfekantu.czujnikGórnegoPoziomu := 0;
   tor[1].zbiornikDezynfekantu.czujnikGórnegoPoziomu := 50;
   tor[2].zbiornikDezynfekantu.czujnikGórnegoPoziomu := 59;
   tor[0].zbiornikDezynfekantu.temperatura := 0;
   tor[1].zbiornikDezynfekantu.temperatura := 5;
   tor[2].zbiornikDezynfekantu.temperatura := 6;
   tor[0].zbiornikDezynfekantu.poziomAnalogowy := 0;
   tor[1].zbiornikDezynfekantu.poziomAnalogowy := 15;
   tor[2].zbiornikDezynfekantu.poziomAnalogowy := 16;
   tor[0].zbiornikDezynfekantu.czujnikwłazu := 0;
   tor[1].zbiornikDezynfekantu.czujnikwłazu := 53;
   tor[2].zbiornikDezynfekantu.czujnikwłazu := 62;
   tor[0..2].zbiornikDezynfekantu.zbiornikDezynfekantu.czujnikDolnegoPoziomu := 0;
   tor[0..2].zbiornikDezynfekantu.zbiornikDezynfekantu.czujnikGórnegoPoziomu := 0;
   tor[0..2].zbiornikDezynfekantu.zbiornikDezynfekantu.temperatura := 0;
   tor[0..2].zbiornikDezynfekantu.zbiornikDezynfekantu.poziomAnalogowy := 0;
   tor[0..2].zbiornikDezynfekantu.zbiornikDezynfekantu.czujnikwłazu := 0;
   tor[0].zbiornikDezynfekantu_2.czujnikDolnegoPoziomu := 0;
   tor[1].zbiornikDezynfekantu_2.czujnikDolnegoPoziomu := 70;
   tor[2].zbiornikDezynfekantu_2.czujnikDolnegoPoziomu := 0;
   tor[0].zbiornikDezynfekantu_2.czujnikGórnegoPoziomu := 0;
   tor[1].zbiornikDezynfekantu_2.czujnikGórnegoPoziomu := 69;
   tor[2].zbiornikDezynfekantu_2.czujnikGórnegoPoziomu := 0;
   tor[0].zbiornikDezynfekantu_2.temperatura := 0;
   tor[1].zbiornikDezynfekantu_2.temperatura := 7;
   tor[2].zbiornikDezynfekantu_2.temperatura := 0;
   tor[0].zbiornikDezynfekantu_2.poziomAnalogowy := 0;
   tor[1].zbiornikDezynfekantu_2.poziomAnalogowy := 17;
   tor[2].zbiornikDezynfekantu_2.poziomAnalogowy := 0;
   tor[0].zbiornikDezynfekantu_2.czujnikwłazu := 0;
   tor[1].zbiornikDezynfekantu_2.czujnikwłazu := 71;
   tor[2].zbiornikDezynfekantu_2.czujnikwłazu := 0;
   tor[0..2]."-zbiorniki na stacji przygotowania chemii" := FALSE;
   tor[0].zbiorniczekDozowaniaŁugu.czujnikDolnegoPoziomu := 81;
   tor[1..2].zbiorniczekDozowaniaŁugu.czujnikDolnegoPoziomu := 0;
   tor[0..2].zbiorniczekDozowaniaŁugu.czujnikGórnegoPoziomu := 0;
   tor[0..2].zbiorniczekDozowaniaŁugu.temperatura := 0;
   tor[0..2].zbiorniczekDozowaniaŁugu.poziomAnalogowy := 0;
   tor[0..2].zbiorniczekDozowaniaŁugu.czujnikwłazu := 0;
   tor[0..2].zbiorniczekDozowaniaŁugu.zbiornikDezynfekantu.czujnikDolnegoPoziomu := 0;
   tor[0..2].zbiorniczekDozowaniaŁugu.zbiornikDezynfekantu.czujnikGórnegoPoziomu := 0;
   tor[0..2].zbiorniczekDozowaniaŁugu.zbiornikDezynfekantu.temperatura := 0;
   tor[0..2].zbiorniczekDozowaniaŁugu.zbiornikDezynfekantu.poziomAnalogowy := 0;
   tor[0..2].zbiorniczekDozowaniaŁugu.zbiornikDezynfekantu.czujnikwłazu := 0;
   tor[0].zbiorniczekDozowaniaKwasu.czujnikDolnegoPoziomu := 43;
   tor[1..2].zbiorniczekDozowaniaKwasu.czujnikDolnegoPoziomu := 0;
   tor[0..2].zbiorniczekDozowaniaKwasu.czujnikGórnegoPoziomu := 0;
   tor[0..2].zbiorniczekDozowaniaKwasu.temperatura := 0;
   tor[0..2].zbiorniczekDozowaniaKwasu.poziomAnalogowy := 0;
   tor[0..2].zbiorniczekDozowaniaKwasu.czujnikwłazu := 0;
   tor[0..2].zbiorniczekDozowaniaKwasu.zbiornikDezynfekantu.czujnikDolnegoPoziomu := 0;
   tor[0..2].zbiorniczekDozowaniaKwasu.zbiornikDezynfekantu.czujnikGórnegoPoziomu := 0;
   tor[0..2].zbiorniczekDozowaniaKwasu.zbiornikDezynfekantu.temperatura := 0;
   tor[0..2].zbiorniczekDozowaniaKwasu.zbiornikDezynfekantu.poziomAnalogowy := 0;
   tor[0..2].zbiorniczekDozowaniaKwasu.zbiornikDezynfekantu.czujnikwłazu := 0;
   tor[0].zbiorniczekDozowanieDezynfekantu.czujnikDolnegoPoziomu := 0;
   tor[1].zbiorniczekDozowanieDezynfekantu.czujnikDolnegoPoziomu := 52;
   tor[2].zbiorniczekDozowanieDezynfekantu.czujnikDolnegoPoziomu := 61;
   tor[0..2].zbiorniczekDozowanieDezynfekantu.czujnikGórnegoPoziomu := 0;
   tor[0..2].zbiorniczekDozowanieDezynfekantu.temperatura := 0;
   tor[0..2].zbiorniczekDozowanieDezynfekantu.poziomAnalogowy := 0;
   tor[0..2].zbiorniczekDozowanieDezynfekantu.czujnikwłazu := 0;
   tor[0..2].zbiorniczekDozowanieDezynfekantu.zbiornikDezynfekantu.czujnikDolnegoPoziomu := 0;
   tor[0..2].zbiorniczekDozowanieDezynfekantu.zbiornikDezynfekantu.czujnikGórnegoPoziomu := 0;
   tor[0..2].zbiorniczekDozowanieDezynfekantu.zbiornikDezynfekantu.temperatura := 0;
   tor[0..2].zbiorniczekDozowanieDezynfekantu.zbiornikDezynfekantu.poziomAnalogowy := 0;
   tor[0..2].zbiorniczekDozowanieDezynfekantu.zbiornikDezynfekantu.czujnikwłazu := 0;
   tor[0..2]."--nalinii" := FALSE;
   tor[0].temperaturaZaWymiennikiem := 0;
   tor[1].temperaturaZaWymiennikiem := 10;
   tor[2].temperaturaZaWymiennikiem := 11;
   tor[0].przepływomierzZaWymiennikiem := 0;
   tor[1].przepływomierzZaWymiennikiem := 106;
   tor[2].przepływomierzZaWymiennikiem := 107;
   tor[0].temperaturaNaPowrocie := 0;
   tor[1].temperaturaNaPowrocie := 8;
   tor[2].temperaturaNaPowrocie := 9;
   tor[0].przewodnośćNaPowrocie := 0;
   tor[1].przewodnośćNaPowrocie := 13;
   tor[2].przewodnośćNaPowrocie := 12;
   tor[0].czujnikPrzepływuNaPowrocie := 0;
   tor[1].czujnikPrzepływuNaPowrocie := 101;
   tor[2].czujnikPrzepływuNaPowrocie := 102;
   tor[0..2]."-naobiekcie" := FALSE;
   tor[0..2].czujnikDolnegoPoziomuwZbiornikuDrenowanym := 0;
   tor[0..2]."-przygotowaniechemii" := FALSE;
   tor[0].pompkaDozowaniaŁuguwLinię := 29;
   tor[1].pompkaDozowaniaŁuguwLinię := 109;
   tor[2].pompkaDozowaniaŁuguwLinię := 0;
   tor[0].pompkaDozowaniaKwasuwLinię := 99;
   tor[1].pompkaDozowaniaKwasuwLinię := 108;
   tor[2].pompkaDozowaniaKwasuwLinię := 0;
   tor[0].pompkaDozowaniaDezynfekantuwLinię := 0;
   tor[1].pompkaDozowaniaDezynfekantuwLinię := 97;
   tor[2].pompkaDozowaniaDezynfekantuwLinię := 98;
   tor[0..1].zawórDozowaniaLuguwLinię := 0;
   tor[2].zawórDozowaniaLuguwLinię := 78;
   tor[0..1].zawórDozowaniaKwasuwLinię := 0;
   tor[2].zawórDozowaniaKwasuwLinię := 41;
   tor[0].zawórDozowaniaDezynfekantuwLinię := 0;
   tor[1].zawórDozowaniaDezynfekantuwLinię := 49;
   tor[2].zawórDozowaniaDezynfekantuwLinię := 58;
   tor[0..2].czujnikPrzepływuDozowanegoŁugu := 0;
   tor[0..2].czujnikPrzepływuDozowanegoKwasu := 0;
   tor[0].czujnikPrzepływuDozowanegoDezynfekantu := 0;
   tor[1].czujnikPrzepływuDozowanegoDezynfekantu := 103;
   tor[2].czujnikPrzepływuDozowanegoDezynfekantu := 104;
   tor[0..2].PrzepływomierzDozowanejChemii := 0;
END_DATA_BLOCK
